{attribute 'GeneratedUsingTerminal: EK1100-0000-0018'}
{attribute addProperty BoxType "EK1100-0000-0018"}
{attribute addProperty Id "Beckhoff_ELM36xxEK1122Beckhoff_ELM36xxEK1122_91B399322A_0001_ELM3602_0000_0017ELM3602_B416BFEF50A_0002_ELM3602_0000_0018ELM3602_B416BFEF50A_0003_ELM3602_0002_0016ELM3602_B416BFEF50A_0004_ELM3602_0002_0017ELM3602_B416BFEF50A_0005_ELM3602_0002_0018ELM3602_B416BFEF50A_0006_ELM3604_0000_0017ELM3604_9E251EA472A_0007_ELM3604_0000_0018ELM3604_9E251EA472A_0008_ELM3604_0002_0016ELM3604_9E251EA472A_0009_ELM3604_0002_0017ELM3604_9E251EA472A_0010_ELM3604_0002_0018ELM3604_9E251EA472"}
{attribute addProperty CRC "746352555"}
{attribute addProperty Size "612"}
TYPE Beckhoff_ELM36xx_2C7C6FAB EXTENDS EK1100_1FC0878B :
STRUCT
	{attribute addProperty Name "Beckhoff_ELM36xxEK1122"}
	{attribute addProperty PreviousPort "Beckhoff ELM36xx : B"}
	Beckhoff_ELM36xxEK1122 : Beckhoff_ELM36xxEK1122_91B39932;
	{attribute addProperty Name "A_0001_ELM3602_0000_0017"}
	{attribute addProperty PreviousPort "Beckhoff ELM36xxEK1122 : C"}
	A_0001_ELM3602_0000_0017 : ELM3602_B416BFEF;
	{attribute addProperty Name "A_0002_ELM3602_0000_0018"}
	{attribute addProperty PreviousPort "A_0001(ELM3602-0000-0017) : B"}
	A_0002_ELM3602_0000_0018 : ELM3602_B416BFEF;
	{attribute addProperty Name "A_0003_ELM3602_0002_0016"}
	{attribute addProperty PreviousPort "A_0002(ELM3602-0000-0018) : B"}
	A_0003_ELM3602_0002_0016 : ELM3602_B416BFEF;
	{attribute addProperty Name "A_0004_ELM3602_0002_0017"}
	{attribute addProperty PreviousPort "A_0003(ELM3602-0002-0016) : B"}
	A_0004_ELM3602_0002_0017 : ELM3602_B416BFEF;
	{attribute addProperty Name "A_0005_ELM3602_0002_0018"}
	{attribute addProperty PreviousPort "A_0004(ELM3602-0002-0017) : B"}
	A_0005_ELM3602_0002_0018 : ELM3602_B416BFEF;
	{attribute addProperty Name "A_0006_ELM3604_0000_0017"}
	{attribute addProperty PreviousPort "A_0005(ELM3602-0002-0018) : B"}
	A_0006_ELM3604_0000_0017 : ELM3604_9E251EA4;
	{attribute addProperty Name "A_0007_ELM3604_0000_0018"}
	{attribute addProperty PreviousPort "A_0006(ELM3604-0000-0017) : B"}
	A_0007_ELM3604_0000_0018 : ELM3604_9E251EA4;
	{attribute addProperty Name "A_0008_ELM3604_0002_0016"}
	{attribute addProperty PreviousPort "A_0007(ELM3604-0000-0018) : B"}
	A_0008_ELM3604_0002_0016 : ELM3604_9E251EA4;
	{attribute addProperty Name "A_0009_ELM3604_0002_0017"}
	{attribute addProperty PreviousPort "A_0008(ELM3604-0002-0016) : B"}
	A_0009_ELM3604_0002_0017 : ELM3604_9E251EA4;
	{attribute addProperty Name "A_0010_ELM3604_0002_0018"}
	{attribute addProperty PreviousPort "A_0009(ELM3604-0002-0017) : B"}
	A_0010_ELM3604_0002_0018 : ELM3604_9E251EA4;
END_STRUCT
END_TYPE

(* stored: Version 1.2.0.0, ProductVersion 3.1.4024.9
   DUT Beckhoff_ELM36xx_2C7C6FAB: Id {5376d5f2-80b6-4696-b036-ca35f263dfa3} *)
